Yaskawa INFORM job: aruba_cylinder_program_no_t.JBI

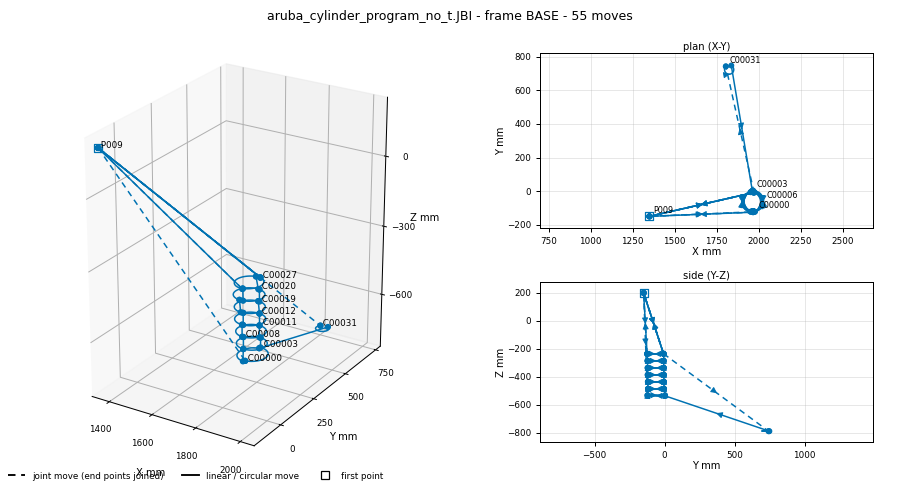
[picture p0: tool path of aruba_cylinder_program_no_t.JBI in frame BASE, 55 of 70 moves have a stored position in this frame; points joined in program order, loops and branches not executed]
/JOB
//NAME aruba_cylinder_program_no_t
//POS
///NPOS 64,0,64,1,0,1
///TOOL 0
///POSTYPE BASE
///RECTAN
///RCONF 0,0,0,0,0,0,0,0,0,0,0,0,0,0,0,0,0,0,0,0,0,0,0,0
C00000=1977.600,-122.295,-530.338,90.0000,-90.0000,5.0000
C00001=1977.600,-122.295,-530.338,90.0000,-90.0000,5.0000
C00002=2028.960,-52.590,-530.338,175.0000,-89.9999,5.0000
C00003=1967.680,3.293,-530.338,-90.0000,-90.0000,5.0000
C00004=1972.400,-4.204,-484.971,-90.0000,-90.0000,5.0000
C00005=1972.400,-4.204,-484.971,-90.0000,-90.0000,5.0000
C00006=2026.850,-62.229,-484.971,175.0000,-89.9999,5.0000
C00007=1967.770,-119.093,-484.971,90.0000,-90.0000,5.0000
C00008=1968.010,-119.618,-434.971,90.0000,-90.0000,5.0000
C00009=1968.010,-119.618,-434.971,90.0000,-90.0000,5.0000
C00010=2023.080,-62.471,-434.971,175.0000,-89.9999,5.0000
C00011=1967.760,-4.723,-434.971,-90.0000,-90.0000,5.0000
C00012=1967.740,-5.412,-384.971,-90.0000,-90.0000,5.0000
C00013=1967.740,-5.412,-384.971,-90.0000,-90.0000,5.0000
C00014=2020.570,-67.817,-384.971,175.0000,-89.9999,5.0000
C00015=1967.670,-120.531,-384.971,90.0000,-90.0000,5.0000
C00016=1967.810,-120.855,-334.971,90.0000,-90.0000,5.0000
C00017=1967.810,-120.855,-334.971,90.0000,-90.0000,5.0000
C00018=2018.500,-67.526,-334.971,175.0000,-89.9999,5.0000
C00019=1967.910,-6.129,-334.971,-90.0000,-90.0000,5.0000
C00020=1967.720,-6.629,-284.971,-90.0000,-90.0000,5.0000
C00021=1967.720,-6.629,-284.971,-90.0000,-90.0000,5.0000
C00022=2017.270,-67.184,-284.971,175.0000,-89.9999,5.0000
C00023=1967.820,-121.635,-284.971,90.0000,-90.0000,5.0000
C00024=1968.570,-124.679,-234.229,90.0000,-90.0000,5.0000
C00025=1968.570,-124.679,-234.229,90.0000,-90.0000,5.0000
C00026=2012.270,-62.782,-234.229,175.0000,-89.9999,5.0000
C00027=1972.510,-7.978,-234.229,-90.0000,-90.0000,5.0000
C00028=1972.510,-7.978,-234.229,-90.0000,-90.0000,5.0000
C00029=1972.510,-7.978,-234.229,-90.0000,-90.0000,5.0000
C00030=1972.510,-7.978,-234.229,-90.0000,-90.0000,5.0000
C00031=1804.730,742.635,-787.417,180.0000,-60.0000,0.0000
C00032=1804.730,742.635,-787.417,180.0000,-60.0000,0.0000
C00033=1842.270,744.534,-787.417,180.0000,-60.0000,0.0000
C00034=1837.320,747.876,-787.417,180.0000,-60.0000,0.0000
C00035=1962.440,2.876,-534.971,-90.0000,-90.0000,5.0000
C00036=1962.440,2.876,-534.971,-90.0000,-90.0000,5.0000
C00037=1913.370,-57.215,-534.971,5.0000,-89.9999,5.0000
C00038=1967.650,-122.308,-534.971,90.0000,-90.0000,5.0000
C00039=1967.530,-119.186,-484.971,90.0000,-90.0000,5.0000
C00040=1967.530,-119.186,-484.971,90.0000,-90.0000,5.0000
C00041=1911.440,-57.261,-484.971,5.0000,-89.9999,5.0000
C00042=1967.180,-4.100,-484.971,-90.0000,-90.0000,5.0000
C00043=1967.330,-4.775,-434.971,-90.0000,-90.0000,5.0000
C00044=1967.330,-4.775,-434.971,-90.0000,-90.0000,5.0000
C00045=1909.210,-57.201,-434.971,5.0000,-89.9999,5.0000
C00046=1962.660,-120.079,-434.971,90.0000,-90.0000,5.0000
C00047=1962.830,-120.781,-384.971,90.0000,-90.0000,5.0000
C00048=1962.830,-120.781,-384.971,90.0000,-90.0000,5.0000
C00049=1904.340,-62.615,-384.971,5.0000,-89.9999,5.0000
C00050=1967.460,-5.164,-384.971,-90.0000,-90.0000,5.0000
C00051=1962.280,-5.488,-334.971,-90.0000,-90.0000,5.0000
C00052=1962.280,-5.488,-334.971,-90.0000,-90.0000,5.0000
C00053=1903.400,-62.352,-334.971,5.0000,-89.9999,5.0000
C00054=1957.370,-121.635,-334.971,90.0000,-90.0000,5.0000
C00055=1952.630,-122.531,-284.971,90.0000,-90.0000,5.0000
C00056=1952.630,-122.531,-284.971,90.0000,-90.0000,5.0000
C00057=1899.440,-62.425,-284.971,5.0000,-89.9999,5.0000
C00058=1962.460,-6.002,-284.971,-90.0000,-90.0000,5.0000
C00059=1952.270,-5.936,-235.586,-90.0000,-90.0000,5.0000
C00060=1952.270,-5.936,-235.586,-90.0000,-90.0000,5.0000
C00061=1905.150,-58.315,-235.586,5.0000,-89.9999,5.0000
C00062=1966.580,-125.367,-235.586,90.0000,-90.0000,5.0000
C00063=1966.580,-125.367,-235.586,90.0000,-90.0000,5.0000
///POSTYPE PULSE
///PULSE
EC00000=0
EC00001=0
EC00002=0
EC00003=0
EC00004=0
EC00005=0
EC00006=0
EC00007=0
EC00008=0
EC00009=0
EC00010=0
EC00011=0
EC00012=0
EC00013=0
EC00014=0
EC00015=0
EC00016=0
EC00017=0
EC00018=0
EC00019=0
EC00020=0
EC00021=0
EC00022=0
EC00023=0
EC00024=0
EC00025=0
EC00026=0
EC00027=0
EC00028=0
EC00029=0
EC00030=0
EC00031=0
EC00032=0
EC00033=0
EC00034=0
EC00035=0
EC00036=0
EC00037=0
EC00038=0
EC00039=0
EC00040=0
EC00041=0
EC00042=0
EC00043=0
EC00044=0
EC00045=0
EC00046=0
EC00047=0
EC00048=0
EC00049=0
EC00050=0
EC00051=0
EC00052=0
EC00053=0
EC00054=0
EC00055=0
EC00056=0
EC00057=0
EC00058=0
EC00059=0
EC00060=0
EC00061=0
EC00062=0
EC00063=0
///POSTYPE BASE
///RECTAN
///RCONF 1,0,0,0,0,0,0,0,0,0,0,0,0,0,0,0,0,0,0,0,0,0,0,0
P00009=1350.000,-150.000,200.000,-180.0000,-45.0000,0.0000
///POSTYPE PULSE
///PULSE
EX00000=0
//INST
///DATE 2023/05/21 16:51
///ATTR SC,RW,RJ
////FRAME BASE
///GROUP1 RB1,ST1
NOP
MOVJ P009 EX000 VJ=15.00
MOVJ P009 VJ=15.00
MOVJ C00000 EC00000 VJ=15.00
MOVC C00001 EC00001 V=50.0
MOVC C00002 EC00002 V=50.0
MOVC C00003 EC00003 V=50.0
MOVL C00004 EC00004 V=50.0
MOVC C00005 EC00005 V=50.0
MOVC C00006 EC00006 V=50.0
MOVC C00007 EC00007 V=50.0
MOVL C00008 EC00008 V=50.0
MOVC C00009 EC00009 V=50.0
MOVC C00010 EC00010 V=50.0
MOVC C00011 EC00011 V=50.0
MOVL C00012 EC00012 V=50.0
MOVC C00013 EC00013 V=50.0
MOVC C00014 EC00014 V=50.0
MOVC C00015 EC00015 V=50.0
MOVL C00016 EC00016 V=50.0
MOVC C00017 EC00017 V=50.0
MOVC C00018 EC00018 V=50.0
MOVC C00019 EC00019 V=50.0
MOVL C00020 EC00020 V=50.0
MOVC C00021 EC00021 V=50.0
MOVC C00022 EC00022 V=50.0
MOVC C00023 EC00023 V=50.0
MOVL C00024 EC00024 V=50.0
MOVC C00025 EC00025 V=50.0
MOVC C00026 EC00026 V=50.0
MOVC C00027 EC00027 V=50.0
MOVJ P009 VJ=15.00
MOVL C00028 EC00028 V=50.0
MOVJ P009 VJ=15.00
MOVL C00029 EC00029 V=50.0
MOVJ P009 VJ=15.00
MOVL C00030 EC00030 V=50.0
MOVJ C00031 EC00031 VJ=15.00
MOVC C00032 EC00032 V=50.0
MOVC C00033 EC00033 V=50.0
MOVC C00034 EC00034 V=50.0
MOVL C00035 EC00035 V=50.0
MOVC C00036 EC00036 V=50.0
MOVC C00037 EC00037 V=50.0
MOVC C00038 EC00038 V=50.0
MOVL C00039 EC00039 V=50.0
MOVC C00040 EC00040 V=50.0
MOVC C00041 EC00041 V=50.0
MOVC C00042 EC00042 V=50.0
MOVL C00043 EC00043 V=50.0
MOVC C00044 EC00044 V=50.0
MOVC C00045 EC00045 V=50.0
MOVC C00046 EC00046 V=50.0
MOVL C00047 EC00047 V=50.0
MOVC C00048 EC00048 V=50.0
MOVC C00049 EC00049 V=50.0
MOVC C00050 EC00050 V=50.0
MOVL C00051 EC00051 V=50.0
MOVC C00052 EC00052 V=50.0
MOVC C00053 EC00053 V=50.0
MOVC C00054 EC00054 V=50.0
MOVL C00055 EC00055 V=50.0
MOVC C00056 EC00056 V=50.0
MOVC C00057 EC00057 V=50.0
MOVC C00058 EC00058 V=50.0
MOVL C00059 EC00059 V=50.0
MOVC C00060 EC00060 V=50.0
MOVC C00061 EC00061 V=50.0
MOVC C00062 EC00062 V=50.0
MOVJ P009 VJ=15.00
MOVL C00063 EC00063 V=50.0
END
